(* IEC 61131-3 sources: plc_generation_empirical_study/datasets/task_bank_v0_2/tasks/C01_B15_composite/negative_control, 1 file *)

(* ---- NC1.st ---- *)
FUNCTION_BLOCK C01_B15_composite
VAR_INPUT
    A_AutoMode : BOOL;
    A_AutoDemand : BOOL;
    A_ManualDemand : BOOL;
    A_SafetyOK : BOOL;
    A_Inhibit : BOOL;
    B_S1 : BOOL;
    B_S2 : BOOL;
    B_S3 : BOOL;
    SubsystemBEnable : BOOL;
    CrossReset : BOOL;
END_VAR
VAR_OUTPUT
    A_Command : BOOL;
    A_Blocked : BOOL;
    B_Vote : BOOL;
    B_Unanimous : BOOL;
    CrossReady : BOOL;
    CrossBlocked : BOOL;
END_VAR

A_Command := ((A_AutoMode AND A_AutoDemand) OR ((NOT A_AutoMode) AND A_ManualDemand))
           AND A_SafetyOK AND (NOT A_Inhibit);
A_Blocked := ((A_AutoMode AND A_AutoDemand) OR ((NOT A_AutoMode) AND A_ManualDemand))
           AND ((NOT A_SafetyOK) OR A_Inhibit);

IF CrossReset THEN
    CrossReady := FALSE;
ELSIF A_Command THEN
    CrossReady := FALSE;
END_IF;
CrossBlocked := SubsystemBEnable AND (NOT CrossReady);

IF SubsystemBEnable AND CrossReady THEN
    B_Vote := (B_S1 AND B_S2) OR (B_S1 AND B_S3) OR (B_S2 AND B_S3);
    B_Unanimous := (B_S1 AND B_S2 AND B_S3) OR ((NOT B_S1) AND (NOT B_S2) AND (NOT B_S3));
ELSE
    B_Vote := FALSE;
    B_Unanimous := FALSE;
END_IF;

END_FUNCTION_BLOCK
